(* PLC project Unnamed, Unknown Unnamed 1 *)
(* stored: creationDateTime 2013-01-29T14:01:00, modificationDateTime 2017-06-08T15:59:13 *)

(* Set input REAL type variable in modbus holding registers *)
FUNCTION SET_HOLDING_REAL : INT
  VAR_INPUT
    ADDR : UINT;
  END_VAR
  VAR_INPUT
    IN_REAL : REAL;
  END_VAR

                    
                     {{
                     #include <stdint.h>
                     typedef uint32_t u32;
                     typedef uint16_t u16;
                     typedef uint8_t u8;
                     extern u8 setU16Holding (u32 adr, u16 value);
                     u32 value = *(u32 *)(&IN_REAL);
                     u16 high = value;
                     u16 low = value >> 16;
                     SET_HOLDING_REAL = setU16Holding(ADDR, high);
                     SET_HOLDING_REAL = setU16Holding(ADDR + 1, low);
                     }}
                    
                    
END_FUNCTION

(* Set input WORD type variable in modbus holding register *)
FUNCTION SET_HOLDING_WORD : INT
  VAR_INPUT
    ADDR : UINT;
  END_VAR
  VAR_INPUT
    IN_WORD : WORD;
  END_VAR

                    
                     {{
                     #include <stdint.h>
                     typedef uint32_t u32;
                     typedef uint16_t u16;
                     typedef uint8_t u8;
                     extern u8 setU16Holding (u32 adr, u16 value);
                     SET_HOLDING_WORD = setU16Holding(ADDR, IN_WORD);
                     }}
                    
                    
END_FUNCTION

(* Set input WORD type variable in modbus holding register *)
FUNCTION SET_HOLDING_LONG : INT
  VAR_INPUT
    ADDR : UINT;
  END_VAR
  VAR_INPUT
    IN_DWORD : DWORD;
  END_VAR

                    
                     {{
                     #include <stdint.h>
                     typedef uint32_t u32;
                     typedef uint16_t u16;
                     typedef uint8_t u8;
                     extern u8 setU16Holding (u32 adr, u16 value);
                     u16 high = IN_DWORD;
                     u16 low = IN_DWORD >> 16;
                     setU16Holding(ADDR, IN_DWORD);
                     SET_HOLDING_LONG = setU16Holding(ADDR + 1, (IN_DWORD >> 16));
                     }}
                    
                    
END_FUNCTION

(* Return REAL type variable from modbus holding registers *)
FUNCTION GET_HOLDING_REAL : REAL
  VAR_INPUT
    ADDR : UINT;
  END_VAR

                        
                     {{
                     #include <stdint.h>
                     typedef uint32_t u32;
                     typedef uint16_t u16;
                     typedef uint8_t u8;
                     extern u16 getU16Holding (u32 adr);
                     u16 higth, low;
                     u32 value;
                     low = getU16Holding(ADDR);
                     higth = getU16Holding(ADDR + 1);
                     value = (higth<< 16) | (low);
                     GET_HOLDING_REAL = *(float *)(& value);
                     }}
                    
                    
END_FUNCTION

(* Return WORD type variable from modbus holding register *)
FUNCTION GET_HOLDING_WORD : WORD
  VAR_INPUT
    ADDR : UINT;
  END_VAR

                        
                     {{
                     #include <stdint.h>
                     typedef uint32_t u32;
                     typedef uint16_t u16;
                     typedef uint8_t u8;
                     extern u16 getU16Holding (u32 adr);
                     GET_HOLDING_WORD = getU16Holding(ADDR);
                     }}
                    
                    
END_FUNCTION

(* Return WORD type variable from modbus holding register *)
FUNCTION GET_HOLDING_LONG : DWORD
  VAR_INPUT
    ADDR : UINT;
  END_VAR

                        
                     {{
                     #include <stdint.h>
                     typedef uint32_t u32;
                     typedef uint16_t u16;
                     typedef uint8_t u8;
                     extern u16 getU16Holding (u32 adr);
                     u16 high= getU16Holding(ADDR);
                     u16 low = getU16Holding(ADDR + 1);
                     GET_HOLDING_LONG = (low << 16) | high;
                     }}
                    
                    
END_FUNCTION

(* Set input WORD type variable in modbus input register *)
FUNCTION SET_INPUT_WORD : INT
  VAR_INPUT
    ADDR : UINT;
  END_VAR
  VAR_INPUT
    IN_WORD : WORD;
  END_VAR

                        
                     {{
                     #include <stdint.h>
                     typedef uint32_t u32;
                     typedef uint16_t u16;
                     typedef uint8_t u8;
                     extern u8 setU16Input(u32 adr, u16 value);
                     SET_INPUT_WORD = setU16Input(ADDR, IN_WORD);
                     }}
                    
                    
END_FUNCTION

(* Return WORD type variable from modbus input register *)
FUNCTION GET_INPUT_WORD : WORD
  VAR_INPUT
    ADDR : UINT;
  END_VAR

                        
                     {{
                     #include <stdint.h>
                     typedef uint32_t u32;
                     typedef uint16_t u16;
                     typedef uint8_t u8;
                     extern u16 getU16Input (u32 adr);
                     GET_INPUT_WORD = getU16Input(ADDR);
                     }}
                    
                    
END_FUNCTION

(* Set input WORD type variable in modbus coil register *)
FUNCTION SET_COIL : INT
  VAR_INPUT
    ADDR : UINT;
  END_VAR
  VAR_INPUT
    COIL_VALUE : BOOL;
  END_VAR

                        
                     {{
                     #include <stdint.h>
                     typedef uint32_t u32;
                     typedef uint16_t u16;
                     typedef uint8_t u8;
                     extern u8 setCoil (u32 adr, u8 value);
                     SET_COIL = setCoil(ADDR, COIL_VALUE);
                     }}
                    
                    
END_FUNCTION

FUNCTION GET_COIL : BOOL
  VAR_INPUT
    ADDR : UINT;
  END_VAR

                        
                     {{
                     #include <stdint.h>
                     typedef uint32_t u32;
                     typedef uint16_t u16;
                     typedef uint8_t u8;
                     extern u8 getCoil (u32 adr);
                     GET_COIL = getCoil(ADDR);
                     }}
                    
                    
END_FUNCTION

(* Return BOOL type variable from modbus input register *)
FUNCTION SET_DISC : INT
  VAR_INPUT
    ADDR : UINT;
  END_VAR
  VAR_INPUT
    DISC_VALUE : BOOL;
  END_VAR

                        
                     {{
                     #include <stdint.h>
                     typedef uint32_t u32;
                     typedef uint16_t u16;
                     typedef uint8_t u8;
                     extern u8 setDisc (u32 adr, u8 value);
                     SET_DISC = setDisc(ADDR, DISC_VALUE);
                     }}
                    
                    
END_FUNCTION

FUNCTION GET_DISC : BOOL
  VAR_INPUT
    ADDR : UINT;
  END_VAR

                        
                     {{
                     #include <stdint.h>
                     typedef uint32_t u32;
                     typedef uint16_t u16;
                     typedef uint8_t u8;
                     extern u8 getDisc (u32 adr);
                     GET_DISC = getDisc(ADDR);
                     }}
                    
                    
END_FUNCTION
